{attribute 'qualified_only'}
{attribute 'strict'}
TYPE E_StationState :
(
	IDLE := 0,
	DETECTION,
	FILLING,
	COMPLETE,
	ERROR
);
END_TYPE

(* stored: Version 1.1.0.1, ProductVersion 3.1.4024.16
   DUT E_StationState: Id {b6f418c6-8e48-49cc-9b39-fcddbf1d2d7b} *)
